(* Logix 5000 project; controller AnalogIO_Shared vendor 1 type 14 code 155 rev 36.11; software revision 36.00 *)

TASK MainTask (continuous, watchdog 500 ms) : MainProgram

MODULES
   Local : vendor 1 type 14 code 155 (PointIO 0, rev 36.11)
       : 1734-IE2V (PointIO 2, rev 3.1, Input RPI 80 ms)
       : 1734-OE2V (PointIO 3, rev 3.1, Output RPI 80 ms)
      Discrete_IO : Embedded (PointIO 1, rev 36.11, Output RPI 20 ms)
END_MODULES

PROGRAM MainProgram   (* main routine MotorControlla *)
VAR
   centripetalClock : FBD_TIMER;
   i_AnalogVoltageInput : ALIAS FOR Local:2:I.Ch0Data;
   i_GreenPB : ALIAS FOR Local:1:I.Data.0;
   i_MilkTemp : ALIAS FOR Local:2:I.Ch1Data;
   i_MixerHeight : ALIAS FOR Local:2:I.Ch0Data;
   i_NightModeButton : ALIAS FOR Local:1:I.Data.3;
   i_RedPB_StopButton : ALIAS FOR Local:1:I.Data.1;
   i_Turnkey : ALIAS FOR Local:1:I.Data.2;
   mixingClock : FBD_TIMER;
   myClock : FBD_TIMER;
   o_AnalogVoltageOutput : ALIAS FOR Local:3:O.Ch1Data;
   o_CentrAccel : ALIAS FOR Local:1:O.Data.10;
   o_heater : ALIAS FOR Local:1:O.Data.14;
   o_homogenizer : ALIAS FOR Local:1:O.Data.15;
   o_mixer : ALIAS FOR Local:1:O.Data.12;
   o_pump1 : ALIAS FOR Local:1:O.Data.11;
   o_pump2 : ALIAS FOR Local:1:O.Data.13;
   pasteurizeClock : FBD_TIMER;
   Pause : DINT;
   s_Centripetal : DINT;
   s_Heater : DINT;
   s_Homogenizer : DINT;
   s_Mixing : DINT;
   s_Pasteurize : DINT;
   s_Pump2_WaitForNoFlow : DINT;
   s_PumpIntoMixer : DINT;
   s_PumpOutOfMixer : DINT;
   s_WaitForStart : DINT;
   Start : DINT;
   StateCurrent : DINT;
   StateNext : DINT;
   StatePrev : DINT;
END_VAR

ROUTINE MotorControlla   (* structured text *)
   RTOR(centripetalClock);
   RTOR(pasteurizeClock);
   RTOR(mixingClock);
   
   // Set clock preset
   if(s:fs) then
   	s_WaitForStart := 0;
   	s_Centripetal := 1;
   	s_PumpIntoMixer := 2;
   	s_Mixing := 3;
   	s_PumpOutOfMixer := 4;
   	s_Heater := 5;
   	s_Pasteurize := 6;
   	s_Pump2_WaitForNoFlow := 7;
   	s_Homogenizer := 8;
   
   	centripetalClock.TimerEnable := 0;
   	pasteurizeClock.TimerEnable := 0;
   	mixingClock.TimerEnable := 0;
   	StateCurrent := s_WaitForStart;
   end_if;
   
   //Timer allows move to next state
   if(myClock.DN) then
   	myClock.Reset := 1;
   	StateCurrent := StateNext;
   else
   	myClock.Reset := 0;
   end_if;
   
   // Pause button
   if ((not i_RedPB_StopButton)) then
   	Pause := 1;
   	Start := 0;
   end_if;
   
   // Start button
   if (i_GreenPB) then
   	Start := 1;
   	Pause := 0;
   end_if;
   
   //State logic
   //s_WaitForStart
   if (StateCurrent = s_WaitForStart) then
   	StatePrev := StateCurrent;
   	o_CentrAccel := 0;
   	o_pump1 := 0;
   	o_mixer := 0;
   	o_pump2 := 0;
   	o_heater := 0;
   	o_homogenizer := 0;
   	if (not(i_GreenPB)) then
   		StateCurrent := s_WaitForStart;
   	else
   		StateCurrent := s_Centripetal;
   
   		o_CentrAccel := 0;
   		o_pump1 := 0;
   		o_mixer := 0;
   		o_pump2 := 0;
   		o_heater := 0;
   		o_homogenizer := 0;
   		StateNext := s_WaitForStart;
   	end_if;
   end_if;
   
   //s_Centripetal
   if (StateCurrent = s_Centripetal) then
   	centripetalClock.PRE := 10000;
   	centripetalClock.TimerEnable := 1;
   	StatePrev := StateCurrent;
   	o_CentrAccel := 1;
   	o_pump1 := 0;
   	o_mixer := 0;
   	o_pump2 := 0;
   	o_heater := 0;
   	o_homogenizer := 0;
   	if (not(centripetalClock.DN)) then
   		StateCurrent := s_Centripetal;
   	else
   		StateCurrent := s_PumpIntoMixer;
   
   
   		o_pump1 := 0;
   		o_mixer := 0;
   		o_pump2 := 0;
   		o_heater := 0;
   		o_CentrAccel := 0;
   		o_homogenizer := 0;
   		StateNext := s_PumpIntoMixer;
   	end_if;
   end_if;
   
   //s_PumpIntoMixer
   if (StateCurrent = s_PumpIntoMixer) then
   	StatePrev := StateCurrent;
   	o_pump1 := 1;
   	o_CentrAccel := 0;
   	o_mixer := 0;
   	o_pump2 := 0;
   	o_heater := 0;
   	o_homogenizer := 0;
   	if (i_MixerHeight < 6400) then //6.4V = 80% mixer height if 8V = 100%
   		StateCurrent := s_PumpIntoMixer;
   	else
   		StateCurrent := s_Mixing;
   
   		o_pump1 := 0;
   		o_CentrAccel := 0;
   		o_mixer := 0;
   		o_pump2 := 0;
   		o_heater := 0;
   		o_homogenizer := 0;
   		StateNext := s_Mixing;
   	end_if;
   end_if;
   
   //s_Mixing
   if (StateCurrent = s_Mixing) then
   	mixingClock.PRE := 5000;
   	mixingClock.TimerEnable := 1;
   	o_mixer := 1;
   	o_CentrAccel := 0;
   	o_pump1 := 0;
   	o_pump2 := 0;
   	o_heater := 0;
   	o_homogenizer := 0;
   	StatePrev := StateCurrent;
   	if (not(mixingClock.DN)) then
   		StateCurrent := s_Mixing;
   	else
   		StateCurrent := s_PumpOutOfMixer;
   
   		o_CentrAccel := 0;
   		o_pump1 := 0;
   		o_pump2 := 0;
   		o_heater := 0;
   		o_homogenizer := 0;
   		o_mixer := 0;
   		StateNext := s_Mixing;
   	end_if;
   end_if;
   
   //s_PumpOutOfMixer
   if (StateCurrent = s_PumpOutOfMixer) then
   	StatePrev := StateCurrent;
   	o_pump2 := 1;
   	o_CentrAccel := 0;
   	o_pump1 := 0;
   	o_mixer := 0;
   	o_heater := 0;
   	o_homogenizer := 0;
   	if (not(i_MixerHeight < 80)) then //0.08V = 1% of mixer height if 8V is 100%
   		StateCurrent := s_PumpOutOfMixer;
   	else
   		StateCurrent := s_Heater;
   
   		o_CentrAccel := 0;
   		o_pump1 := 0;
   		o_mixer := 0;
   		o_heater := 0;
   		o_homogenizer := 0;
   		o_pump2 := 0;
   		StateNext := s_Heater;
   	end_if;
   end_if;
   
   //s_Heater
   if (StateCurrent = s_Heater) then
   	StatePrev := StateCurrent;
   	o_heater := 1;
   	o_CentrAccel := 0;
   	o_pump1 := 0;
   	o_pump2 := 0;
   	o_mixer := 0;
   	o_homogenizer := 0;
   	if (not(i_MilkTemp > 8100)) then //8.1V = 162F if 10V = 200F
   		StateCurrent := s_Heater;
   	else
   		StateCurrent := s_Pasteurize;
   
   		o_CentrAccel := 0;
   		o_heater := 0;
   		o_pump1 := 0;
   		o_pump2 := 0;
   		o_mixer := 0;
   		o_homogenizer := 0;
   		StateNext := s_Pasteurize;
   	end_if;
   end_if;
   
   //s_Pasteurize
   if (StateCurrent = s_Pasteurize) then
   	StatePrev := StateCurrent;
   	pasteurizeClock.PRE := 15500;
   	pasteurizeClock.TimerEnable := 1;
   	o_CentrAccel := 0;
   	o_pump1 := 0;
   	o_pump2 := 0;
   	o_mixer := 0;
   	o_heater := 0;
   	o_homogenizer := 0;
   	if (not(pasteurizeClock.DN)) then
   		StateCurrent := s_Pasteurize;
   	elsif (i_Turnkey) then
   		StateCurrent := s_Pasteurize;
   	else
   		StateCurrent := s_Pump2_WaitForNoFlow;
   
   		o_CentrAccel := 0;
   		o_pump1 := 0;
   		o_pump2 := 0;
   		o_mixer := 0;
   		o_heater := 0;
   		o_homogenizer := 0;
   		StateNext := s_Pump2_WaitForNoFlow;
   	end_if;
   end_if;
   
   //s_Pump2_WaitForNoFlow
   if (StateCurrent = s_Pump2_WaitForNoFlow) then
   	StatePrev := StateCurrent;
   	o_pump2 := 1;
   	o_CentrAccel := 0;
   	o_pump1 := 0;
   	o_mixer := 0;
   	o_heater := 0;
   	o_homogenizer := 0;
   	if (not(i_Turnkey)) then
   		StateCurrent := s_Pump2_WaitForNoFlow;
   	else
   		StateCurrent := s_Homogenizer;
   
   		o_CentrAccel := 0;
   		o_pump1 := 0;
   		o_mixer := 0;
   		o_heater := 0;
   		o_homogenizer := 0;
   		o_pump2 := 0;
   		StateNext := s_Pump2_WaitForNoFlow;
   	end_if;
   end_if;
   
   //s_Homogenizer
   if (StateCurrent = s_Homogenizer) then
   	StatePrev := StateCurrent;
   	o_homogenizer := 1;
   	o_CentrAccel := 0;
   	o_pump1 := 0;
   	o_pump2 := 0;
   	o_mixer := 0;
   	o_heater := 0;
   	if (not(i_NightModeButton)) then //NightModeButton = Homogenizer finished button
   		StateCurrent := s_Homogenizer;
   	else
   		StateCurrent := s_WaitForStart;
   
   		o_CentrAccel := 0;
   		o_pump1 := 0;
   		o_pump2 := 0;
   		o_mixer := 0;
   		o_heater := 0;
   		o_homogenizer := 0;
   		StateNext := s_WaitForStart;
   	end_if;
   end_if;
   
   
END_ROUTINE
END_PROGRAM
